PROGRAM P_TpKommunikation
VAR
	
END_VAR

//Netzwerk 1:
//F_AuswertungBefehlstastenVonTP(); nur noch in den Tasten-Events

//Netzwerk 2:
F_AnzeigeNiedriegePrio();

//Netzwerk 3:
//F_SignaldauerVonTastleuchte_MaschEinAuswerten();

//Netzwerk 4:
F_SAFETY_AnzeigenHohePrio_Neu();

END_PROGRAM

(* stored: Version 1.1.0.1, ProductVersion 3.1.4024.3
   POU P_TpKommunikation: Id {b93ec95b-18ca-44f3-8e6d-35b2b63f1e5b}, SpecialFunc None *)
